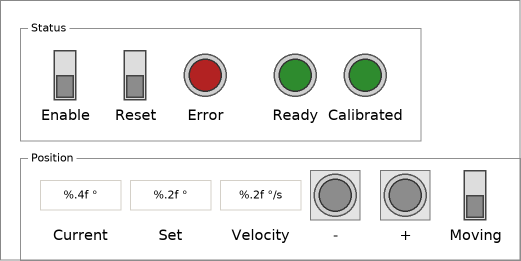
VISUALIZATION Elevation  // 521x261
    GroupBox (20,20 401x121), "Status"
        DipSwitch (20,30 50x50), variable: MAIN.ElevationControl.enable, behaviour: TOGGLE, style: Switch-DipSwitch-Gray
        DipSwitch (90,30 50x50), variable: MAIN.ElevationControl.reset, behaviour: TOGGLE, style: Switch-DipSwitch-Gray
        Label (0,80 91x30), "Enable"
        Label (80,80 71x30), "Reset"
        Lamp1 (160,30 50x50), variable: MAIN.ElevationControl.error, style: Lamp-Lamp1-Red
        Label (160,80 51x30), "Error"
        Lamp1 (250,30 50x50), variable: MAIN.ElevationControl.Ready, style: Lamp-Lamp1-Green
        Lamp1 (320,30 50x50), variable: MAIN.ElevationControl.Calibrated, style: Lamp-Lamp1-Green
        Label (250,80 51x30), "Ready"
    Label (330,100 71x30), "Calibrated"
    GroupBox (20,150 501x111), "Position"
        Label (20,70 81x30), "Current"
        Label (350,70 71x30), "+"
        Label (420,70 71x30), "Moving"
        Textfield (20,30 81x30), "%.4f °", text variable: MAIN.ElevationControl.actualPosition
        Label (110,70 81x30), "Set"
        Textfield (110,30 81x30), "%.2f °", text variable: MAIN.ElevationControl.position
            OnMouseClick: write the text variable via InputWithLimits, min MAIN.DerotatorControl.min_position, max MAIN.DerotatorControl.max_position
        PushSwitch (290,20 50x50), variable: MAIN.ElevationControl.down, behaviour: TAP, style: Switch-PushSwitch-Gray
        Label (280,70 71x30), "-"
        PushSwitch (360,20 50x50), variable: MAIN.ElevationControl.up, behaviour: TAP, style: Switch-PushSwitch-Gray
        DipSwitch (430,20 50x50), variable: MAIN.ElevationControl.MoveAxis, behaviour: TOGGLE, style: Switch-DipSwitch-Gray
    Label (220,220 81x30), "Velocity"
    Textfield (220,180 81x30), "%.2f °/s", text variable: MAIN.ElevationControl.velocity
        OnMouseClick: write the text variable via InputWithLimits, min MAIN.DerotatorControl.min_position, max MAIN.DerotatorControl.max_position
END_VISUALIZATION

(* stored: Version 1.1.0.1, ProductVersion 3.1.4026.8
   Visu Elevation: Id {4b29d921-8ee2-4942-802b-58d68324ce04} *)
